{attribute 'qualified_only'}
{attribute 'strict'}
{attribute 'to_string'}
//Pathing Enum
TYPE E_TankBundleNumber :
(
	Bundle_Tank_1:=1,Bundle_Tank_2:=2,Bundle_Tank_3:=3,Bundle_Tank_4:=4
);
END_TYPE

(* stored: Version 1.1.0.1
   DUT E_TankBundleNumber: Id {ef76c0a8-7186-48ea-b729-43d2c2cbd167} *)
